PROGRAM F20_HandScanner
VAR
	fbHandScannerAddress					: FB_HandScannerAddress;
	fbHandScannerCtrl						: ARRAY[1..cMAX_HAND_SCANNERS] OF FB_HandScannerCtrl;
	tmpBarcode								: T_MaxString; (*Left for commissioning*)

(*variables to be removed if IO will be defined*)
{library private}
(***************************Terminal States Diagnostic********************************)

	(*istEtherCATMasterState					: ST_CX_EtherCATMasterState;*)
	iaEtherCATSlaveState					: ARRAY [0..cMAX_ETHERCAT_SLAVES] OF UINT;

	inDummyEL6001PortNo					: UINT;
	istDummyHandScannerCOMPortDataIn		: EL6InData22B;
	qstDummyHandScannerCOMPortDataOut		: EL6OutData22B;
	nTMP:UDINT;
END_VAR

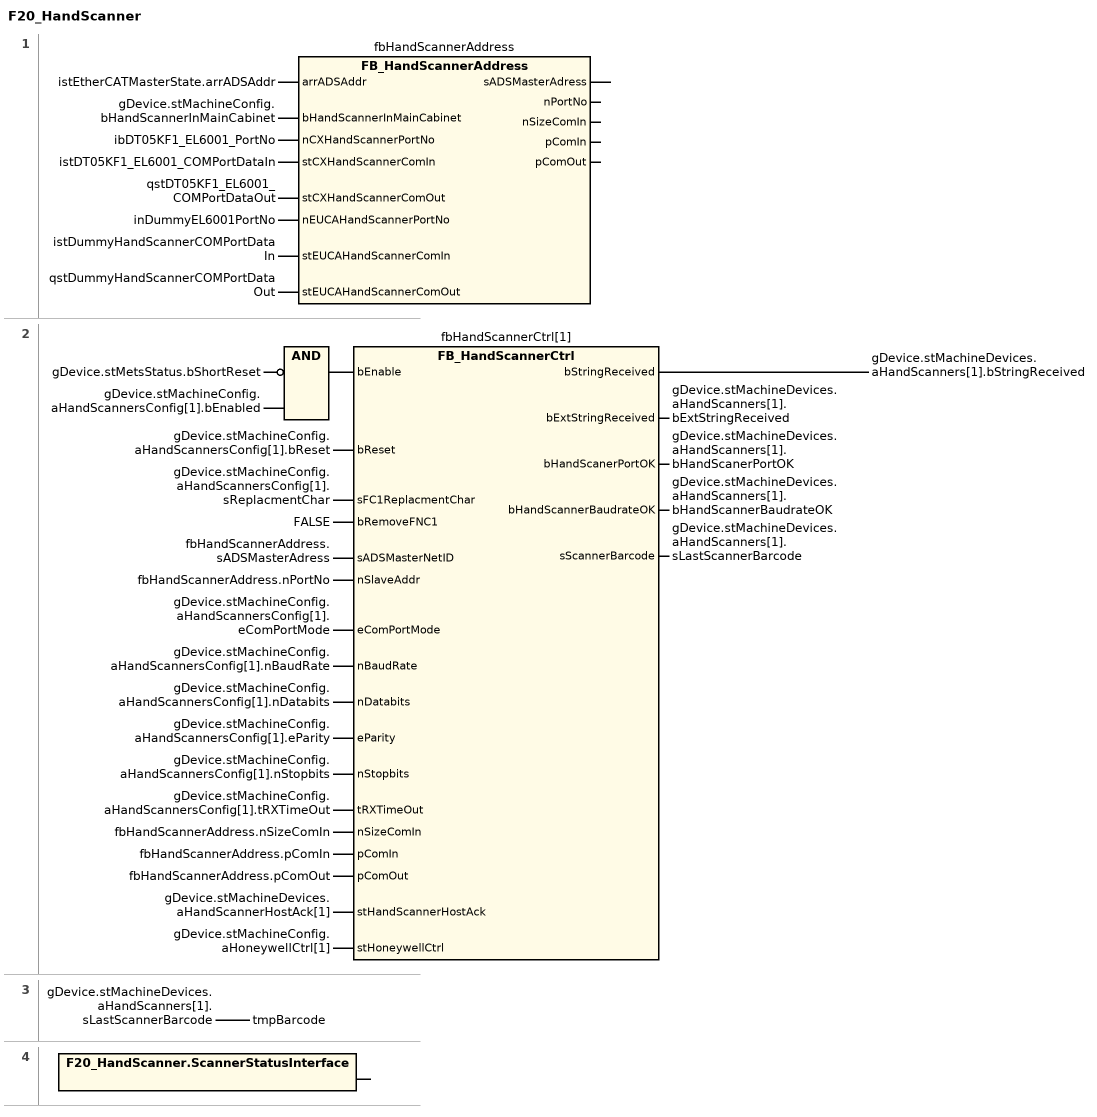
// NETWORK 1
fbHandScannerAddress(
    arrADSAddr := istEtherCATMasterState.arrADSAddr,
    bHandScannerInMainCabinet := gDevice.stMachineConfig.bHandScannerInMainCabinet,
    nCXHandScannerPortNo := ibDT05KF1_EL6001_PortNo,
    stCXHandScannerComIn := istDT05KF1_EL6001_COMPortDataIn,
    stCXHandScannerComOut := qstDT05KF1_EL6001_COMPortDataOut,
    nEUCAHandScannerPortNo := inDummyEL6001PortNo,
    stEUCAHandScannerComIn := istDummyHandScannerCOMPortDataIn,
    stEUCAHandScannerComOut := qstDummyHandScannerCOMPortDataOut); // FB_HandScannerAddress

// NETWORK 2
fbHandScannerCtrl[1](
    bEnable := NOT gDevice.stMetsStatus.bShortReset AND gDevice.stMachineConfig.aHandScannersConfig[1].bEnabled,
    bReset := gDevice.stMachineConfig.aHandScannersConfig[1].bReset,
    sFC1ReplacmentChar := gDevice.stMachineConfig.aHandScannersConfig[1].sReplacmentChar,
    bRemoveFNC1 := FALSE,
    sADSMasterNetID := fbHandScannerAddress.sADSMasterAdress,
    nSlaveAddr := fbHandScannerAddress.nPortNo,
    eComPortMode := gDevice.stMachineConfig.aHandScannersConfig[1].eComPortMode,
    nBaudRate := gDevice.stMachineConfig.aHandScannersConfig[1].nBaudRate,
    nDatabits := gDevice.stMachineConfig.aHandScannersConfig[1].nDatabits,
    eParity := gDevice.stMachineConfig.aHandScannersConfig[1].eParity,
    nStopbits := gDevice.stMachineConfig.aHandScannersConfig[1].nStopbits,
    tRXTimeOut := gDevice.stMachineConfig.aHandScannersConfig[1].tRXTimeOut,
    nSizeComIn := fbHandScannerAddress.nSizeComIn,
    pComIn := fbHandScannerAddress.pComIn,
    pComOut := fbHandScannerAddress.pComOut,
    stHandScannerHostAck := gDevice.stMachineDevices.aHandScannerHostAck[1],
    stHoneywellCtrl := gDevice.stMachineConfig.aHoneywellCtrl[1],
    bExtStringReceived => gDevice.stMachineDevices.aHandScanners[1].bExtStringReceived,
    bHandScanerPortOK => gDevice.stMachineDevices.aHandScanners[1].bHandScanerPortOK,
    bHandScannerBaudrateOK => gDevice.stMachineDevices.aHandScanners[1].bHandScannerBaudrateOK,
    sScannerBarcode => gDevice.stMachineDevices.aHandScanners[1].sLastScannerBarcode); // FB_HandScannerCtrl
gDevice.stMachineDevices.aHandScanners[1].bStringReceived := fbHandScannerCtrl[1].bStringReceived;

// NETWORK 3
tmpBarcode := gDevice.stMachineDevices.aHandScanners[1].sLastScannerBarcode;

// NETWORK 4
F20_HandScanner.ScannerStatusInterface();

ACTION ScannerStatusInterface:
gHMI.aHoneywellStatusHMI[1].bHandScanerPortOK	:= gDevice.stMachineDevices.aHandScanners[1].bHandScanerPortOK;
gHMI.aHoneywellStatusHMI[1].bHandScannerBaudrateOK	:= gDevice.stMachineDevices.aHandScanners[1].bHandScannerBaudrateOK;
gHMI.aHoneywellStatusHMI[1].sLastScannerBarcode		:= gDevice.stMachineDevices.aHandScanners[1].sLastScannerBarcode;
END_ACTION

END_PROGRAM

(* stored: Version 1.1.0.1
   POU F20_HandScanner: Id {09052dcf-54ea-4801-9dce-29969ca60c0d}, SpecialFunc None
   Action ScannerStatusInterface: Id {151a2d2f-4f4c-467c-8f0d-d4f65d79e937} *)
